// TIA Portal V21 export
DATA_BLOCK "块_1_DB_3"   // DB6
// stored: InstanceOfName 块_1, InstanceOfType FB
"块_1"
   // VAR_INPUT
   //    in1 : Bool;
   //    in2 : Bool;
   // END_VAR
   // VAR_OUTPUT
   //    out1 : Bool;
   // END_VAR
BEGIN
END_DATA_BLOCK
